(* IEC 61131-3 sources: virtual-plc/crates/plc-compiler/fuzz/corpus/fuzz_parse, 3 files *)

(* ---- control.st ---- *)
PROGRAM Control
VAR
    i : INT := 0;
    x : INT;
END_VAR
    IF i > 10 THEN
        x := 1;
    ELSIF i < 0 THEN
        x := -1;
    ELSE
        x := 0;
    END_IF;

    CASE i OF
        0: x := 100;
        1, 2: x := 200;
    ELSE
        x := 999;
    END_CASE;

    FOR i := 0 TO 10 DO
        x := x + 1;
    END_FOR;

    WHILE i < 20 DO
        i := i + 1;
    END_WHILE;
END_PROGRAM

(* ---- minimal.st ---- *)
PROGRAM X
VAR
    a : INT;
END_VAR
    a := 1;
END_PROGRAM

(* ---- types.st ---- *)
PROGRAM Types
VAR
    b : BOOL := TRUE;
    i : INT := -100;
    ui : UINT := 100;
    r : REAL := 3.14;
    s : STRING := 'test';
END_VAR
    b := NOT b;
    i := i + 1;
END_PROGRAM
